// TIA Portal V17 export
// export: Created 2024-01-30T08:49:11.7589483Z, ExportSetting WithDefaults, DisplayName Totally Integrated Automation Portal, DisplayVersion V17 Update 6, DisplayName TIA Portal Openness, DisplayVersion V17 Update 6, DisplayName TIA Portal Version Control Interface, DisplayVersion V17, DisplayName STEP 7 Professional, DisplayVersion V17 Update 6, DisplayName STEP 7 Safety, DisplayVersion V17 Update 6, DisplayName WinCC Advanced, DisplayVersion V17 Update 6
FUNCTION_BLOCK "B.05847_FFB"   // FB3, LAD
{ S7_Optimized_Access := 'TRUE' }
VERSION : 0.1
// stored: AutoNumber true, IsIECCheckEnabled false, IsRetainMemResEnabled false, MemoryReserve 100, SetENOAutomatically false, UDAEnableTagReadback false
BEGIN

REGION Network 1: FESTO_CMMT_ST
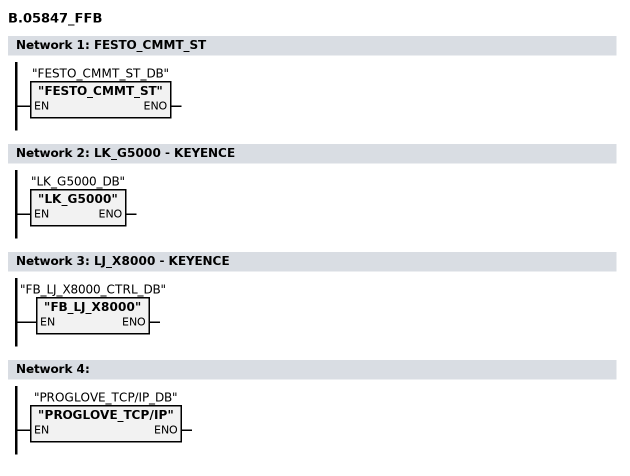
   RUNG wire#powerrail
      "FESTO_CMMT_ST_DB"()
   END_RUNG
   // the same network as SCL:
   "FESTO_CMMT_ST_DB"();   // "FESTO_CMMT_ST"
END_REGION

REGION Network 2: LK_G5000 - KEYENCE
   RUNG wire#powerrail
      "LK_G5000_DB"()
   END_RUNG
   // the same network as SCL:
   "LK_G5000_DB"();   // "LK_G5000"
END_REGION

REGION Network 3: LJ_X8000 - KEYENCE
   RUNG wire#powerrail
      "FB_LJ_X8000_CTRL_DB"()
   END_RUNG
   // the same network as SCL:
   "FB_LJ_X8000_CTRL_DB"();   // "FB_LJ_X8000"
END_REGION

REGION Network 4
   RUNG wire#powerrail
      "PROGLOVE_TCP/IP_DB"()
   END_RUNG
   // the same network as SCL:
   "PROGLOVE_TCP/IP_DB"();   // "PROGLOVE_TCP/IP"
END_REGION
END_FUNCTION_BLOCK
